// TIA Portal V20 export
// export: Created 2025-12-01T14:57:45.5090629Z, ExportSetting None, DisplayName Totally Integrated Automation Portal, DisplayVersion V20 Update 3, DisplayName TIA Portal Openness, DisplayVersion V20 Update 3, DisplayName TIA Portal Version Control Interface, DisplayVersion V20 Update 3, DisplayName STEP 7 Professional, DisplayVersion V20 Update 3, DisplayName STEP 7 Safety, DisplayVersion V20 Update 2, DisplayName WinCC Basic/Comfort/Advanced, DisplayVersion V20 Update 3, DisplayName WinCC Professional, DisplayVersion V20 Update 3, DisplayName WinCC Unified, DisplayVersion V20 Update 3
FUNCTION "FC889_Obtener_ValorDelAtributo_ULint" : Void   // FC889, LAD
TITLE = "ObtemerValorAtributo" - Convertir a Doble Entero una String
{ S7_Optimized_Access := 'FALSE' }
AUTHOR : TRACKING
NAME : 20130301
VERSION : 3.0
// stored: AutoNumber false, SetENOAutomatically false
   VAR_INPUT
      DB_String : Word;   // DB donde esta la String
      OffsetIni : UInt;   // Numero de byte de la String donde empieza
   END_VAR
   VAR_OUTPUT
      Valor : ULInt;   // Valor de la Conversion
   END_VAR
   VAR_TEMP
      PunteroDB : DWord;   // Puntero al DB de la String
      NumDB : Word;   // Numero de DB de la String
      OffsetActual : UInt;   // Numero de bytes de la String Actual
      siguiente_digito : UInt;
      TEMP_Valor : ULInt;
   END_VAR
BEGIN

REGION Network 1 (SCL): inicializaciones
   // inicialización de los valores de trabajo

   #TEMP_Valor := 0;
   #NumDB := #DB_String;
   #OffsetActual := #OffsetIni;

   //
END_REGION

NETWORK
TITLE = Cuerpo de la Funcion
// - Calcula el Puntero al Caracter a Convertir
// - Se mira si es Numero
// - Obteniendo el Nuevo Valor de la Conversion
// - Pasar al siguiente Caracter
// ----------------------------------------------------------------------------------------
// Calcula el Puntero al Caracter a Convertir

InicioBucle:OPN   DB [#NumDB];
      L     #OffsetActual;
      SLD   3;
      T     #PunteroDB;

// ----------------------------------------------------------------------------------------
// Se mira si es numero

      L     DBB [#PunteroDB];
      L     '0';
      <I;
      JC    Final;
      L     DBB [#PunteroDB];
      L     '9';
      >I;
      JC    Final;


NETWORK
TITLE = 

      L     DBB [#PunteroDB];  // Quito la parte Alta del Byte Leido
      L     W#16#F;  // Es como restar w#16#30
      AD;
      T     #siguiente_digito;



REGION Network 4 (SCL): sumarle el siguiente digito
   #TEMP_Valor := (#TEMP_Valor *10)+ #siguiente_digito;
END_REGION

NETWORK
TITLE = 

// ----------------------------------------------------------------------------------------
// Pasar al siguiente caracter

      L     #OffsetActual;  // Continuo para ver si el siguiente es digito
      L     1;
      +I;
      T     #OffsetActual;
      JU    InicioBucle;


Final:NOP   0;


REGION Network 6 (SCL): Valor de la Conversion
   #Valor := #TEMP_Valor;
   "DB209_Reg_Etquetas_Esp_Activa".Reg_Etiqueta[1].CDB := #Valor;
END_REGION
END_FUNCTION
